Fanuc KAREL source: KO00053.KL

PROGRAM KO00053
%NOLOCKGROUP
%ENVIRONMENT MIR
VAR
  P1: XYZWPR
  P2: XYZWPR
  F: BOOLEAN
  OUT: POSITION
BEGIN
  F = TRUE
  OUT = MIRROR(P1, P2, F)
END KO00053
